PROGRAM prg_TrappenhuisautomaatTijdsinstelling
VAR
END_VAR

END_PROGRAM

(* stored: Version 1.1.0.1, ProductVersion 3.1.4024.15
   POU prg_TrappenhuisautomaatTijdsinstelling: Id {fec349af-33a3-4bce-b25c-3eeceaf35561}, SpecialFunc None *)
